FUNCTION And4 : I_BoolValue
VAR_INPUT
	value1 : I_BoolValue;
	value2 : I_BoolValue;
	value3 : I_BoolValue;
	value4 : I_BoolValue;
END_VAR
VAR
	p : POINTER TO FB_BooleanExpression;
END_VAR

p := __NEW(FB_BooleanExpression);

p^.Op4(
	operator := E_BooleanOperator.ANDop,
	value1 := value1,
	value2 := value2,
	value3 := value3,
	value4 := value4
);

And4 := p^;

END_FUNCTION

(* stored: Version 1.1.0.1
   POU And4: Id {097e1958-6933-4acc-86cb-af30df9f2525}, SpecialFunc None *)
